// TwinCAT 3 PLC project PLC_Program
// ProgramVersion: 3.1.4024.0
// libraries:
//   Tc2_MC2, * (Beckhoff Automation GmbH)
//   Tc2_Standard, * (Beckhoff Automation GmbH)
//   Tc2_System, * (Beckhoff Automation GmbH)
//   Tc3_Module, * (Beckhoff Automation GmbH)
// project tree:
//   / PlcTask.TcTTO
//   POUs/ MAIN.TcPOU, Motion.TcPOU
// real-time tasks:
//   TASK PlcTask: cycle T#10ms, priority 20, ADS port 350
//   TASK MainTask: cycle T#4ms, priority 1, ADS port 351
//   TASK VISU_TASK: cycle T#1ms, priority 31, ADS port 352
//   TASK EtherCAT_Task: cycle T#1ms, priority ?, ADS port 353
//   TASK PlcTask1: cycle T#10ms, priority 21, ADS port 354
// motion (NC):
//   TASK NC-Task 1 SAF: cycle T#2ms, priority 4, ADS port 501
//   TASK NC-Task 1 SVB: cycle T#10ms, priority 8, ADS port 511
//   AXIS Axis 1 (id 1)
//     General: UnitName=Degree
//     Dynamic: Acceleration=15000, Deceleration=15000, Jerk=225000
//     PositionAreaControl: Range=360
//     OtherSettings: AllowMotionCmdToSlave=true
//     encoder EncType=19
//       EncPara: ScaleFactorNumerator=360, ScaleFactorDenominator=65536, MaxCount=#xffffffff
//     drive DrvType=16
//       DrvPara: MaxCount=#xffffffff, DriveControlDWord=#x00020000
//         Analog: TorqueSetpointScale=10, ScaleFactorActTorque=0.1
//         TimeComp: TaskDelayCycles=1
//     controller CtrType=1
//       CtrPara: PriorControlFactor=1
//         PosDiffControl: Range=500, Time=1
//         Observer: BandWidth=20
// I/O:
//   DEVICE Device 3 (EtherCAT), AmsNetId 5.44.157.108.4.1
//     Drive 1 (Unidrive M700 RFC-S) [Unidrive M700 RFC-S]
// variable links:
//   NC-Task 1 SAF/Axes/Axis 1 <-> Device 3 (EtherCAT)/Drive 1 (Unidrive M700 RFC-S)
//     Drive/Inputs/In/nDcOutputTime <-> InfoData/DcOutputShift
//     Drive/Inputs/In/nState1 <-> Transmit PDO Mapping 3/Status word
//     Drive/Inputs/In/nState2 <-> Transmit PDO Mapping 3/Status word @bit 8
//     Drive/Inputs/In/nState4 @bit 1 <-> WcState/InputToggle
//     Drive/Inputs/In/nState4 <-> WcState/WcState
//     Drive/Outputs/Out/nCtrl1 <-> Receive PDO Mapping 3/Control word
//     Drive/Outputs/Out/nCtrl2 <-> Receive PDO Mapping 3/Control word @bit 8
//     Drive/Outputs/Out/nDataOut1 <-> Receive PDO Mapping 3/Target position
//     Enc/Inputs/In/nDataIn1 <-> Transmit PDO Mapping 3/Position actual value
//     Enc/Inputs/In/nDcInputTime <-> InfoData/DcInputShift
//     Enc/Inputs/In/nState4 @bit 1 <-> WcState/InputToggle
//     Enc/Inputs/In/nState4 <-> WcState/WcState
//   PLC Program/PLC Program Instance <-> NC-Task 1 SAF/Axes/Axis 1
//     PlcTask Inputs/MAIN.Axis1.NcToPlc <-> Outputs/ToPlc
//     PlcTask Outputs/MAIN.Axis1.PlcToNc <-> Inputs/FromPlc

CONFIGURATION PLC_Program
    RESOURCE PLC ON TwinCAT3
        TASK PlcTask(INTERVAL := T#10ms, PRIORITY := 21);
        PROGRAM MAIN WITH PlcTask : MAIN;
        PROGRAM Motion WITH PlcTask : Motion;
    END_RESOURCE
END_CONFIGURATION

// ---- POUs/MAIN.TcPOU
PROGRAM MAIN
VAR
	Axis1: AXIS_REF;
END_VAR

END_PROGRAM

// ---- POUs/Motion.TcPOU
PROGRAM Motion
VAR
	Power : MC_Power;
	Speed : MC_Jog;
	Velocity : MC_MoveVelocity;
	
END_VAR

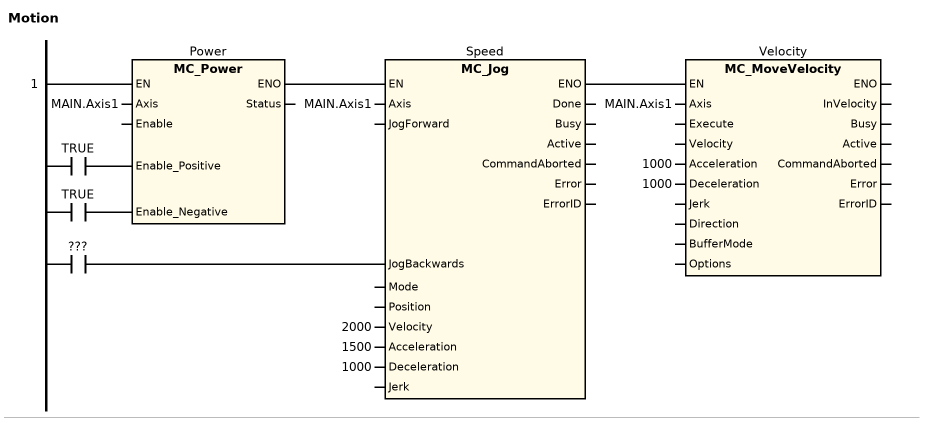
// NETWORK 1
Power(Axis := MAIN.Axis1, Enable_Positive := TRUE, Enable_Negative := TRUE); // MC_Power
Speed(Axis := MAIN.Axis1, Velocity := 2000, Acceleration := 1500, Deceleration := 1000); // MC_Jog
Velocity(Axis := MAIN.Axis1, Acceleration := 1000, Deceleration := 1000); // MC_MoveVelocity

END_PROGRAM
